# EPICS autosave request: support/dac128V/2-4/dac128VApp/Db/8chan_DAC_settings.req
#FILE... 8chan_DAC_settings.req
#USAGE... 8-channel singleDAC.db fields autosave'd.
file "singleDAC_settings.req", P=$(P), D=$(D), N=1
file "singleDAC_settings.req", P=$(P), D=$(D), N=2
file "singleDAC_settings.req", P=$(P), D=$(D), N=3
file "singleDAC_settings.req", P=$(P), D=$(D), N=4
file "singleDAC_settings.req", P=$(P), D=$(D), N=5
file "singleDAC_settings.req", P=$(P), D=$(D), N=6
file "singleDAC_settings.req", P=$(P), D=$(D), N=7
file "singleDAC_settings.req", P=$(P), D=$(D), N=8
